{attribute 'TcGenerated'}
{attribute 'no-analysis'}
{attribute 'linkalways'}
// This function has been automatically generated from the project information.
VAR_GLOBAL CONSTANT
	{attribute 'const_non_replaced'}
	stLibVersion_Project_Title : ST_LibVersion := (iMajor := 0, iMinor := 0, iBuild := 1, iRevision := 1, nFlags := 0, sVersion := '0.0.1.1');
END_VAR

(* stored: Version 1.1.0.1, ProductVersion 3.1.4024.11
   GVL Global_Version: Id {889266fe-3640-0d0d-39e1-17d2f693df42} *)
